(* CODESYS project semaforo_new.project

Project tree, tasks and I/O mapping:
  Device : CODESYS Control Win V3, 3S - Smart Software Solutions GmbH, order no. 305021, version 3.5.10.30
    DeviceApplication
      application Applicazione
        libraries: Standard, * (System)
        task MainTask (cyclic, interval t#20ms, priority 1) calls PLC_PRG
        task VISU_TASK (cyclic, interval 100 ms, priority 31) calls VisuElems.Visu_Prg
        program PLC_PRG [ST]
        visualisation Semaforo_View
  text list GlobalTextList
*)

// Device/DeviceApplication/Applicazione/PLC_PRG
PROGRAM PLC_PRG
VAR
    Red    : BOOL;
    Yellow : BOOL;
    Green  : BOOL;
    state  : INT := 0;
    t      : TON;
END_VAR

CASE state OF
    0:
        Red := TRUE; Yellow := FALSE; Green := FALSE;
        t(IN := TRUE, PT := T#5S);
        IF t.Q THEN
            state := 1;
            t(IN := FALSE);
        END_IF
    1:
        Red := TRUE; Yellow := TRUE; Green := FALSE;
        t(IN := TRUE, PT := T#2S);
        IF t.Q THEN
            state := 2;
            t(IN := FALSE);
        END_IF
    2:
        Red := FALSE; Yellow := FALSE; Green := TRUE;
        t(IN := TRUE, PT := T#5S);
        IF t.Q THEN
            state := 3;
            t(IN := FALSE);
        END_IF
    3:
        Red := FALSE; Yellow := TRUE; Green := FALSE;
        t(IN := TRUE, PT := T#2S);
        IF t.Q THEN
            state := 0;
            t(IN := FALSE);
        END_IF
END_CASE

END_PROGRAM

// Device/DeviceApplication/Applicazione/Semaforo_View
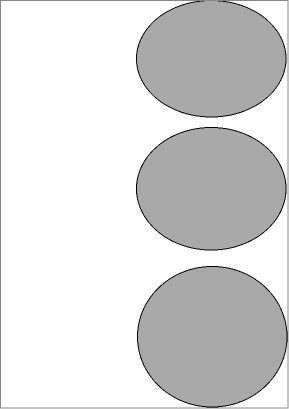
VISUALIZATION Semaforo_View  // 289x409
    Ellipse (136,0 150x117), colour toggle: PLC_PRG.Red
    Ellipse (136,127 150x123), colour toggle: PLC_PRG.Yellow
    Ellipse (137,266 150x141), colour toggle: PLC_PRG.Green
END_VISUALIZATION
